(* IEC 61131-3 sources: AXOpen/src/components.cognex.vision/app/SystemConstants (part 3) *)

    END_VAR
END_CONFIGURATION
